{attribute 'pack_mode' := '2'}
TYPE ST_PackTwo :
STRUCT
	bBoolMember1 : BOOL;
	nDwordMember : DWORD;
	bBoolMember2 : BOOL;
	nLwordMember : LWORD;
END_STRUCT
END_TYPE

(* stored: Version 1.1.0.1, ProductVersion 3.1.4024.13
   DUT ST_PackTwo: Id {a1b2c3d4-0000-4000-8000-000000000002} *)
